(* PLC project PLC, Beckhoff Automation GmbH TwinCAT PLC Control 3.5.13.21 *)
(* stored: creationDateTime 2024-02-17T22:43:25.555054, modificationDateTime 2024-02-17T22:43:25.555054 *)

(* global variable list G *)
{attribute 'qualified_only'}
VAR_GLOBAL CONSTANT
	numAxis: LINT := 128;
	nameStringLength: LINT := 64;
END_VAR
VAR_GLOBAL
END_VAR
